{attribute 'linkalways'} 
{attribute 'no_explicit_call' := 'This FB is a CLASS and must be accessed using methods or properties'}
{attribute 'enable_dynamic_creation'}
FUNCTION_BLOCK Node_F_VN_SetAt_INT EXTENDS VisionNode
VAR
    nElement : _INT(0);
    ipContainer : _ITcVnContainer;
    nIndex : _ULINT(0);
    hrPrev : _HRESULT(S_OK);
    hresult : _HRESULT(S_OK);
END_VAR

METHOD PUBLIC  Clone : I_Node
VAR
	pNode : POINTER TO Node_F_VN_SetAt_INT;
END_VAR
pNode := __NEW(Node_F_VN_SetAt_INT);
Clone := pNode^;
END_METHOD

METHOD FB_init : BOOL
VAR_INPUT
	bInitRetains : BOOL; // if TRUE, the retain variables are initialized (warm start / cold start)
	bInCopyCode : BOOL;  // if TRUE, the instance afterwards gets moved into the copy code (online change)
END_VAR
AddParameter('nElement', nElement);
AddInput('ipContainer', ipContainer);
AddParameter('nIndex', nIndex);
AddInput('hrPrev', hrPrev);
AddOutput('ipContainer', ipContainer);
AddOutput('hresult',hresult);
END_METHOD

METHOD PROTECTED OnExecute
hresult.Value := F_VN_SetAt_INT(
    nElement := nElement.Value,
    ipContainer := ipContainer.Value,
    nIndex := nIndex.Value,
    hrPrev:= hrPrev.Value);
END_METHOD

METHOD PUBLIC PreExecutionCheck
VAR_INPUT
	Check : I_PreExecutionChecks;
END_VAR
Check.IsTrue(ipContainer.IsValid, 'ipContainer must be a valid container');
Check.IsTrue(ipContainer.IsType(TC_GLOBAL_CONST_LIST.ContainerType_Vector_INT), 'ipContainer contains incorrect type');
END_METHOD

END_FUNCTION_BLOCK

(* stored: Version 1.1.0.1, ProductVersion 3.1.4026.13
   POU Node_F_VN_SetAt_INT: Id {87bd9c88-1ef9-4a65-98e3-a26d45f07ed2}, SpecialFunc None
   Folder Constructor: Id {a6a67c7b-30a2-4ed3-ab41-0b8df8da5afa}
   Method Clone: Id {b303309d-de1b-4911-a2a6-85a9cfd174e6}
   Method FB_init: Id {1c590023-19f2-48e1-955d-2fdd0bc03931}
   Method OnExecute: Id {f2039b33-ba98-4f69-bb90-6d4687b2120c}
   Method PreExecutionCheck: Id {f64a4c03-fd2f-4e50-8604-700b8f2c4620} *)
